TYPE ST_Tray_1 :
STRUCT
	{attribute 'OPC.UA.DA' := '1'}
	nCropID : UDINT;
	{attribute 'OPC.UA.DA' := '0'}
	nLineID : UDINT;
	{attribute 'OPC.UA.DA' := '0'}
	nOrderID : UDINT;
	{attribute 'OPC.UA.DA' := '0'}
	nPlantID : UDINT; 
	{attribute 'OPC.UA.DA' := '0'}
	nStack : INT;
	{attribute 'OPC.UA.DA' := '0'}
	nRack : INT;
	{attribute 'OPC.UA.DA' := '0'}
	nLevel : INT;
	{attribute 'OPC.UA.DA' := '0'}
	nRestack : INT;
	
	{attribute 'OPC.UA.DA' := '1'}
	nTrayQuantity: INT;
	{attribute 'OPC.UA.DA' := '1'}
	nTrayNumber: INT;
	
END_STRUCT
END_TYPE

(* stored: Version 1.1.0.1, ProductVersion 3.1.4024.12
   DUT ST_Tray_1: Id {8337bcb3-0bc8-419f-9aa0-adf946e58039} *)
